  Call Extruder(271.09444)
  MoveL 11489 to (229.08, 163.95, 153.89) mm, rotated rx 180 ry 0 rz 180 deg; joints [-30.766, 12.961, 71.357, 80.556, 31.236, -78.992]
  MoveL 11490 to (229.08, 163.95, 153.89) mm, rotated rx 180 ry 0 rz 180 deg; joints [-30.766, 12.961, 71.357, 80.556, 31.236, -78.992]
  Call Extruder(271.20816)
  MoveL 11491 to (228.87, 164, 153.89) mm, rotated rx 180 ry 0 rz 180 deg; joints [-30.781, 12.934, 71.389, 80.571, 31.249, -79.007]
  MoveL 11492 to (228.87, 164, 153.89) mm, rotated rx 180 ry 0 rz 180 deg; joints [-30.781, 12.934, 71.389, 80.571, 31.249, -79.007]
  Call Extruder(271.33358)
  MoveL 11493 to (228.65, 164.04, 153.89) mm, rotated rx -180 ry 0 rz 180 deg; joints [-30.797, 12.904, 71.425, 80.587, 31.264, -79.024]
  MoveL 11494 to (228.65, 164.04, 153.89) mm, rotated rx -180 ry 0 rz 180 deg; joints [-30.797, 12.904, 71.425, 80.587, 31.264, -79.024]
  Call Extruder(271.47056)
  MoveL 11495 to (228.4, 164.09, 153.89) mm, rotated rx 180 ry 0 rz -180 deg; joints [-30.815, 12.872, 71.464, 80.604, 31.281, -79.042]
  MoveL 11496 to (228.4, 164.09, 153.89) mm, rotated rx 180 ry 0 rz -180 deg; joints [-30.815, 12.872, 71.464, 80.604, 31.281, -79.042]
  Call Extruder(271.60692)
  MoveL 11497 to (228.15, 164.14, 153.89) mm, rotated rx -180 ry 0 rz 180 deg; joints [-30.832, 12.839, 71.504, 80.622, 31.297, -79.06]
  MoveL 11498 to (228.15, 164.14, 153.89) mm, rotated rx -180 ry 0 rz 180 deg; joints [-30.832, 12.839, 71.504, 80.622, 31.297, -79.06]
  Call Extruder(271.74268)
  MoveL 11499 to (227.9, 164.19, 153.89) mm, rotated rx 180 ry 0 rz 180 deg; joints [-30.85, 12.806, 71.543, 80.639, 31.313, -79.079]
  MoveL 11500 to (227.9, 164.19, 153.89) mm, rotated rx 180 ry 0 rz 180 deg; joints [-30.85, 12.806, 71.543, 80.639, 31.313, -79.079]
  Call Extruder(271.87783)
  MoveL 11501 to (227.65, 164.24, 153.89) mm, rotated rx 180 ry 0 rz 180 deg; joints [-30.868, 12.773, 71.583, 80.656, 31.329, -79.097]
  MoveL 11502 to (227.65, 164.24, 153.89) mm, rotated rx 180 ry 0 rz 180 deg; joints [-30.868, 12.773, 71.583, 80.656, 31.329, -79.097]
  Call Extruder(272.01237)
  MoveL 11503 to (227.4, 164.29, 153.89) mm, rotated rx 180 ry 0 rz 180 deg; joints [-30.886, 12.74, 71.622, 80.674, 31.346, -79.115]
  MoveL 11504 to (227.4, 164.29, 153.89) mm, rotated rx 180 ry 0 rz 180 deg; joints [-30.886, 12.74, 71.622, 80.674, 31.346, -79.115]
  Call Extruder(272.14629)
  MoveL 11505 to (227.15, 164.34, 153.89) mm, rotated rx 180 ry 0 rz -180 deg; joints [-30.903, 12.708, 71.662, 80.691, 31.362, -79.133]
  MoveL 11506 to (227.15, 164.34, 153.89) mm, rotated rx 180 ry 0 rz -180 deg; joints [-30.903, 12.708, 71.662, 80.691, 31.362, -79.133]
  Call Extruder(272.29416)
  MoveL 11507 to (226.87, 164.39, 153.89) mm, rotated rx 180 ry 0 rz -180 deg; joints [-30.923, 12.671, 71.706, 80.71, 31.38, -79.154]
  MoveL 11508 to (226.87, 164.39, 153.89) mm, rotated rx 180 ry 0 rz -180 deg; joints [-30.923, 12.671, 71.706, 80.71, 31.38, -79.154]
  Call Extruder(272.45590)
  MoveL 11509 to (226.57, 164.44, 153.89) mm, rotated rx 180 ry 0 rz 180 deg; joints [-30.943, 12.63, 71.756, 80.731, 31.399, -79.176]
  MoveL 11510 to (226.57, 164.44, 153.89) mm, rotated rx 180 ry 0 rz 180 deg; joints [-30.943, 12.63, 71.756, 80.731, 31.399, -79.176]
  Call Extruder(272.61691)
  MoveL 11511 to (226.26, 164.49, 153.89) mm, rotated rx -180 ry 0 rz 180 deg; joints [-30.964, 12.588, 71.805, 80.752, 31.418, -79.198]
  MoveL 11512 to (226.26, 164.49, 153.89) mm, rotated rx -180 ry 0 rz 180 deg; joints [-30.964, 12.588, 71.805, 80.752, 31.418, -79.198]
  Call Extruder(272.77720)
  MoveL 11513 to (225.95, 164.54, 153.89) mm, rotated rx 180 ry 0 rz -180 deg; joints [-30.985, 12.547, 71.855, 80.773, 31.437, -79.22]
  MoveL 11514 to (225.95, 164.54, 153.89) mm, rotated rx 180 ry 0 rz -180 deg; joints [-30.985, 12.547, 71.855, 80.773, 31.437, -79.22]
  Call Extruder(272.93675)
  MoveL 11515 to (225.65, 164.58, 153.89) mm, rotated rx -180 ry 0 rz 180 deg; joints [-31.006, 12.506, 71.904, 80.794, 31.456, -79.242]
  MoveL 11516 to (225.65, 164.58, 153.89) mm, rotated rx -180 ry 0 rz 180 deg; joints [-31.006, 12.506, 71.904, 80.794, 31.456, -79.242]
  Call Extruder(273.09558)
  MoveL 11517 to (225.34, 164.63, 153.89) mm, rotated rx -180 ry 0 rz 180 deg; joints [-31.027, 12.465, 71.953, 80.814, 31.475, -79.264]
  MoveL 11518 to (225.34, 164.63, 153.89) mm, rotated rx -180 ry 0 rz 180 deg; joints [-31.027, 12.465, 71.953, 80.814, 31.475, -79.264]
  Call Extruder(273.27425)
  MoveL 11519 to (225, 164.68, 153.89) mm, rotated rx -180 ry 0 rz -180 deg; joints [-31.049, 12.418, 72.01, 80.838, 31.496, -79.289]
  MoveL 11520 to (225, 164.68, 153.89) mm, rotated rx -180 ry 0 rz -180 deg; joints [-31.049, 12.418, 72.01, 80.838, 31.496, -79.289]
  Call Extruder(273.47269)
  MoveL 11521 to (224.61, 164.73, 153.89) mm, rotated rx 180 ry 0 rz 180 deg; joints [-31.074, 12.364, 72.074, 80.864, 31.519, -79.316]
  MoveL 11522 to (224.61, 164.73, 153.89) mm, rotated rx 180 ry 0 rz 180 deg; joints [-31.074, 12.364, 72.074, 80.864, 31.519, -79.316]
  Call Extruder(273.67027)
  MoveL 11523 to (224.22, 164.77, 153.89) mm, rotated rx 180 ry 0 rz 180 deg; joints [-31.1, 12.311, 72.138, 80.89, 31.542, -79.344]
  MoveL 11524 to (224.22, 164.77, 153.89) mm, rotated rx 180 ry 0 rz 180 deg; joints [-31.1, 12.311, 72.138, 80.89, 31.542, -79.344]
  Call Extruder(273.86697)
  MoveL 11525 to (223.84, 164.82, 153.89) mm, rotated rx -180 ry 0 rz 180 deg; joints [-31.125, 12.258, 72.202, 80.915, 31.565, -79.371]
  MoveL 11526 to (223.84, 164.82, 153.89) mm, rotated rx -180 ry 0 rz 180 deg; joints [-31.125, 12.258, 72.202, 80.915, 31.565, -79.371]
  Call Extruder(274.06281)
  MoveL 11527 to (223.45, 164.86, 153.89) mm, rotated rx 180 ry 0 rz -180 deg; joints [-31.15, 12.204, 72.265, 80.941, 31.588, -79.398]
  MoveL 11528 to (223.45, 164.86, 153.89) mm, rotated rx 180 ry 0 rz -180 deg; joints [-31.15, 12.204, 72.265, 80.941, 31.588, -79.398]
  Call Extruder(274.35817)
  MoveL 11529 to (222.86, 164.91, 153.89) mm, rotated rx 180 ry 0 rz 180 deg; joints [-31.186, 12.122, 72.364, 80.979, 31.621, -79.44]
  MoveL 11530 to (222.86, 164.91, 153.89) mm, rotated rx 180 ry 0 rz 180 deg; joints [-31.186, 12.122, 72.364, 80.979, 31.621, -79.44]
  Call Extruder(274.65220)
  MoveL 11531 to (222.27, 164.95, 153.89) mm, rotated rx 180 ry 0 rz 180 deg; joints [-31.222, 12.039, 72.463, 81.018, 31.654, -79.48]
  MoveL 11532 to (222.27, 164.95, 153.89) mm, rotated rx 180 ry 0 rz 180 deg; joints [-31.222, 12.039, 72.463, 81.018, 31.654, -79.48]
  Call Extruder(274.94489)
  MoveL 11533 to (221.68, 165, 153.89) mm, rotated rx -180 ry 0 rz 180 deg; joints [-31.258, 11.956, 72.562, 81.056, 31.687, -79.521]
  MoveL 11534 to (221.68, 165, 153.89) mm, rotated rx -180 ry 0 rz 180 deg; joints [-31.258, 11.956, 72.562, 81.056, 31.687, -79.521]
  Call Extruder(275.51834)
  MoveL 11535 to (220.52, 165.05, 153.89) mm, rotated rx 180 ry 0 rz 180 deg; joints [-31.326, 11.789, 72.76, 81.13, 31.749, -79.601]
  MoveL 11536 to (220.52, 165.05, 153.89) mm, rotated rx 180 ry 0 rz 180 deg; joints [-31.326, 11.789, 72.76, 81.13, 31.749, -79.601]
  Call Extruder(276.23235)
  MoveL 11537 to (219.06, 165.09, 153.89) mm, rotated rx 180 ry 0 rz -180 deg; joints [-31.409, 11.579, 73.01, 81.221, 31.825, -79.699]
  Call Extruder(393.07903)
  MoveL 11538 to (-19.06, 165.09, 153.89) mm, rotated rx -180 ry 0 rz 180 deg; joints [-51.475, -16.768, 100.178, 84.78, 51.776, -81.601]
  Call Extruder(393.50763)
  MoveL 11539 to (-19.94, 165.07, 153.89) mm, rotated rx 180 ry 0 rz 180 deg; joints [-51.582, -16.85, 100.239, 84.782, 51.884, -81.585]
  MoveL 11540 to (-19.94, 165.07, 153.89) mm, rotated rx 180 ry 0 rz 180 deg; joints [-51.582, -16.85, 100.239, 84.782, 51.884, -81.585]
  Call Extruder(394.08108)
  MoveL 11541 to (-21.1, 165.03, 153.89) mm, rotated rx 180 ry 0 rz 180 deg; joints [-51.722, -16.963, 100.321, 84.785, 52.025, -81.562]
  MoveL 11542 to (-21.1, 165.03, 153.89) mm, rotated rx 180 ry 0 rz 180 deg; joints [-51.722, -16.963, 100.321, 84.785, 52.025, -81.562]
  Call Extruder(394.51538)
  MoveL 11543 to (-21.97, 164.98, 153.89) mm, rotated rx 180 ry 0 rz 180 deg; joints [-51.827, -17.048, 100.383, 84.786, 52.131, -81.545]
  MoveL 11544 to (-21.97, 164.98, 153.89) mm, rotated rx 180 ry 0 rz 180 deg; joints [-51.827, -17.048, 100.383, 84.786, 52.131, -81.545]
  Call Extruder(394.80941)
  MoveL 11545 to (-22.56, 164.93, 153.89) mm, rotated rx -180 ry 0 rz -180 deg; joints [-51.897, -17.108, 100.426, 84.786, 52.201, -81.532]
  MoveL 11546 to (-22.56, 164.93, 153.89) mm, rotated rx -180 ry 0 rz -180 deg; joints [-51.897, -17.108, 100.426, 84.786, 52.201, -81.532]
  Call Extruder(395.10477)
  MoveL 11547 to (-23.15, 164.89, 153.89) mm, rotated rx 180 ry 0 rz -180 deg; joints [-51.966, -17.167, 100.469, 84.787, 52.271, -81.52]
  MoveL 11548 to (-23.15, 164.89, 153.89) mm, rotated rx 180 ry 0 rz -180 deg; joints [-51.966, -17.167, 100.469, 84.787, 52.271, -81.52]
  Call Extruder(395.35098)
  MoveL 11549 to (-23.64, 164.84, 153.89) mm, rotated rx 180 ry 0 rz 180 deg; joints [-52.023, -17.217, 100.505, 84.787, 52.329, -81.509]
  MoveL 11550 to (-23.64, 164.84, 153.89) mm, rotated rx 180 ry 0 rz 180 deg; joints [-52.023, -17.217, 100.505, 84.787, 52.329, -81.509]
  Call Extruder(395.54769)
  MoveL 11551 to (-24.03, 164.79, 153.89) mm, rotated rx 180 ry 0 rz 180 deg; joints [-52.067, -17.258, 100.535, 84.787, 52.374, -81.5]
  MoveL 11552 to (-24.03, 164.79, 153.89) mm, rotated rx 180 ry 0 rz 180 deg; joints [-52.067, -17.258, 100.535, 84.787, 52.374, -81.5]
  Call Extruder(395.74526)
  MoveL 11553 to (-24.42, 164.75, 153.89) mm, rotated rx -180 ry 0 rz 180 deg; joints [-52.112, -17.299, 100.564, 84.786, 52.419, -81.491]
  MoveL 11554 to (-24.42, 164.75, 153.89) mm, rotated rx -180 ry 0 rz 180 deg; joints [-52.112, -17.299, 100.564, 84.786, 52.419, -81.491]
  Call Extruder(395.94370)
  MoveL 11555 to (-24.8, 164.7, 153.89) mm, rotated rx 180 ry 0 rz 180 deg; joints [-52.156, -17.339, 100.594, 84.786, 52.464, -81.481]
  MoveL 11556 to (-24.8, 164.7, 153.89) mm, rotated rx 180 ry 0 rz 180 deg; joints [-52.156, -17.339, 100.594, 84.786, 52.464, -81.481]
  Call Extruder(396.14301)
  MoveL 11557 to (-25.19, 164.66, 153.89) mm, rotated rx 180 ry 0 rz -180 deg; joints [-52.2, -17.38, 100.623, 84.785, 52.509, -81.472]
  MoveL 11558 to (-25.19, 164.66, 153.89) mm, rotated rx 180 ry 0 rz -180 deg; joints [-52.2, -17.38, 100.623, 84.785, 52.509, -81.472]
  Call Extruder(396.30184)
  MoveL 11559 to (-25.5, 164.61, 153.89) mm, rotated rx 180 ry 0 rz 180 deg; joints [-52.235, -17.413, 100.647, 84.785, 52.543, -81.465]
  MoveL 11560 to (-25.5, 164.61, 153.89) mm, rotated rx 180 ry 0 rz 180 deg; joints [-52.235, -17.413, 100.647, 84.785, 52.543, -81.465]
  Call Extruder(396.46140)
  MoveL 11561 to (-25.8, 164.56, 153.89) mm, rotated rx 180 ry 0 rz 180 deg; joints [-52.269, -17.447, 100.671, 84.784, 52.578, -81.457]
  MoveL 11562 to (-25.8, 164.56, 153.89) mm, rotated rx 180 ry 0 rz 180 deg; joints [-52.269, -17.447, 100.671, 84.784, 52.578, -81.457]
  Call Extruder(396.62169)
  MoveL 11563 to (-26.11, 164.51, 153.89) mm, rotated rx 180 ry 0 rz 180 deg; joints [-52.303, -17.48, 100.695, 84.783, 52.612, -81.449]
  MoveL 11564 to (-26.11, 164.51, 153.89) mm, rotated rx 180 ry 0 rz 180 deg; joints [-52.303, -17.48, 100.695, 84.783, 52.612, -81.449]
  Call Extruder(396.78271)
  MoveL 11565 to (-26.41, 164.46, 153.89) mm, rotated rx -180 ry 0 rz 180 deg; joints [-52.337, -17.514, 100.719, 84.782, 52.647, -81.441]
  MoveL 11566 to (-26.41, 164.46, 153.89) mm, rotated rx -180 ry 0 rz 180 deg; joints [-52.337, -17.514, 100.719, 84.782, 52.647, -81.441]
  Call Extruder(396.94445)
  MoveL 11567 to (-26.72, 164.41, 153.89) mm, rotated rx 180 ry 0 rz -180 deg; joints [-52.371, -17.547, 100.743, 84.782, 52.681, -81.433]
  MoveL 11568 to (-26.72, 164.41, 153.89) mm, rotated rx 180 ry 0 rz -180 deg; joints [-52.371, -17.547, 100.743, 84.782, 52.681, -81.433]
  Call Extruder(397.10692)
  MoveL 11569 to (-27.02, 164.37, 153.89) mm, rotated rx 180 ry 0 rz 180 deg; joints [-52.405, -17.58, 100.767, 84.781, 52.716, -81.425]
  MoveL 11570 to (-27.02, 164.37, 153.89) mm, rotated rx 180 ry 0 rz 180 deg; joints [-52.405, -17.58, 100.767, 84.781, 52.716, -81.425]
  Call Extruder(397.24085)
  MoveL 11571 to (-27.27, 164.32, 153.89) mm, rotated rx -180 ry 0 rz -180 deg; joints [-52.432, -17.609, 100.788, 84.78, 52.743, -81.418]
  MoveL 11572 to (-27.27, 164.32, 153.89) mm, rotated rx -180 ry 0 rz -180 deg; joints [-52.432, -17.609, 100.788, 84.78, 52.743, -81.418]
  Call Extruder(397.37538)
  MoveL 11573 to (-27.52, 164.27, 153.89) mm, rotated rx 180 ry 0 rz 180 deg; joints [-52.459, -17.637, 100.808, 84.779, 52.771, -81.411]
  MoveL 11574 to (-27.52, 164.27, 153.89) mm, rotated rx 180 ry 0 rz 180 deg; joints [-52.459, -17.637, 100.808, 84.779, 52.771, -81.411]
  Call Extruder(397.51053)
  MoveL 11575 to (-27.77, 164.22, 153.89) mm, rotated rx 180 ry 0 rz 180 deg; joints [-52.486, -17.665, 100.828, 84.778, 52.798, -81.404]
  MoveL 11576 to (-27.77, 164.22, 153.89) mm, rotated rx 180 ry 0 rz 180 deg; joints [-52.486, -17.665, 100.828, 84.778, 52.798, -81.404]
  Call Extruder(397.64629)
  MoveL 11577 to (-28.02, 164.17, 153.89) mm, rotated rx 180 ry 0 rz -180 deg; joints [-52.513, -17.693, 100.848, 84.777, 52.825, -81.397]
  MoveL 11578 to (-28.02, 164.17, 153.89) mm, rotated rx 180 ry 0 rz -180 deg; joints [-52.513, -17.693, 100.848, 84.777, 52.825, -81.397]
  Call Extruder(397.78265)
  MoveL 11579 to (-28.27, 164.12, 153.89) mm, rotated rx 180 ry 0 rz 180 deg; joints [-52.54, -17.722, 100.869, 84.776, 52.853, -81.391]
  MoveL 11580 to (-28.27, 164.12, 153.89) mm, rotated rx 180 ry 0 rz 180 deg; joints [-52.54, -17.722, 100.869, 84.776, 52.853, -81.391]
  Call Extruder(397.86751)
  MoveL 11581 to (-28.42, 164.09, 153.89) mm, rotated rx -180 ry 0 rz 180 deg; joints [-52.556, -17.739, 100.881, 84.775, 52.87, -81.386]
  Set speed (130.0 mm/s)
  MoveL 11582 to (-31.76, 163.31, 153.89) mm, rotated rx 180 ry 0 rz 180 deg; joints [-52.91, -18.13, 101.16, 84.758, 53.229, -81.286]
  Call Extruder(395.86751)
  Set speed (40.0 mm/s)
  MoveL 11583 to (-31.76, 163.31, 153.89) mm, rotated rx 180 ry 0 rz 180 deg; joints [-52.91, -18.13, 101.16, 84.758, 53.229, -81.286]
  Set speed (1000.0 mm/s)
  Call Extruder(-1)
  MoveL 11584 to (-31.76, 163.31, 153.89) mm, rotated rx 180 ry 0 rz 180 deg; joints [-52.91, -18.13, 101.16, 84.758, 53.229, -81.286]
  Call Extruder(0.00000)
  Call M_RunCode(107)
  Call M_RunCode(104)
  Call M_RunCode(84)
  Call M_RunCode(140)

--- program Print3D (robot Denso VS-6577G-B) ---
  Smooth(1)
  Call M_RunCode(107)
  Call M_RunCode(104)
  Set speed (83.3 mm/s)
  Set speed (1000.0 mm/s)
  Set Ref.: Ref002
  Set Tool: nozzle
  Show nozzle
  MoveJ 1 to (0, 34.91, 105) mm, rotated rx 180 ry 0 rz 180 deg; joints [-47.898, 28.981, 154.135, 132.06, 92.089, -2.313]
  MoveL 2 to (0, 34.91, 105) mm, rotated rx 180 ry 0 rz 180 deg; joints [-47.898, 28.981, 154.135, 132.06, 92.089, -2.313]
  MoveL 3 to (0, 34.91, 5) mm, rotated rx 180 ry 0 rz 180 deg; joints [-47.898, 52.446, 146.262, 130.56, 102.419, -14.104]
  MoveL 4 to (0, 34.91, 5) mm, rotated rx 180 ry 0 rz 180 deg; joints [-47.898, 52.446, 146.262, 130.56, 102.419, -14.104]
  Call M_RunCode(109)
  Call M_RunCode(82)
  Call Extruder(0.00000)
  Set speed (130.0 mm/s)
  MoveL 5 to (0, 34.91, 22.22) mm, rotated rx 180 ry 0 rz 180 deg; joints [-47.898, 48.666, 147.922, 130.893, 101.034, -12.462]
  Call Extruder(-2.00000)
  Set speed (40.0 mm/s)
  MoveL 6 to (0, 34.91, 22.22) mm, rotated rx 180 ry 0 rz 180 deg; joints [-47.898, 48.666, 147.922, 130.893, 101.034, -12.462]
  Call Extruder(0.00000)
  Set speed (130.0 mm/s)
  MoveL 7 to (0, 34.91, 22.22) mm, rotated rx 180 ry 0 rz 180 deg; joints [-47.898, 48.666, 147.922, 130.893, 101.034, -12.462]
  Call Extruder(2.00000)
  Set speed (40.0 mm/s)
  MoveL 8 to (0, 34.91, 22.22) mm, rotated rx 180 ry 0 rz 180 deg; joints [-47.898, 48.666, 147.922, 130.893, 101.034, -12.462]
  Set speed (30.0 mm/s)
  MoveL 9 to (0, 34.91, 22.22) mm, rotated rx 180 ry 0 rz 180 deg; joints [-47.898, 48.666, 147.922, 130.893, 101.034, -12.462]
  Call Extruder(209.10557)
  MoveL 10 to (207.51, 34.91, 22.22) mm, rotated rx 180 ry 0 rz 180 deg; joints [-29.348, 52.122, 123.468, 150.579, 86.157, 2.165]
  Call Extruder(210.41057)
  MoveL 11 to (208.82, 34.98, 22.22) mm, rotated rx 180 ry 0 rz -180 deg; joints [-29.266, 52.176, 123.285, 150.657, 86.041, 2.222]
  Call Extruder(213.89122)
  MoveL 12 to (212.3, 35.26, 22.22) mm, rotated rx 180 ry 0 rz 180 deg; joints [-29.038, 52.32, 122.803, 150.874, 85.737, 2.372]
  Call Extruder(214.76022)
  MoveL 13 to (213.16, 35.34, 22.23) mm, rotated rx 180 ry 0 rz 180 deg; joints [-28.98, 52.356, 122.683, 150.929, 85.662, 2.408]
  Call Extruder(215.62924)
  MoveL 14 to (214.01, 35.53, 22.23) mm, rotated rx -180 ry 0 rz -180 deg; joints [-28.913, 52.389, 122.574, 150.993, 85.592, 2.44]
  Call Extruder(219.10988)
  MoveL 15 to (217.4, 36.34, 22.22) mm, rotated rx 180 ry 0 rz 180 deg; joints [-28.639, 52.52, 122.143, 151.256, 85.317, 2.564]
  Call Extruder(219.97888)
  MoveL 16 to (218.25, 36.56, 22.23) mm, rotated rx 180 ry 0 rz -180 deg; joints [-28.569, 52.552, 122.036, 151.323, 85.249, 2.594]
  Call Extruder(220.84782)
  MoveL 17 to (219.06, 36.88, 22.23) mm, rotated rx 180 ry 0 rz 180 deg; joints [-28.492, 52.581, 121.942, 151.398, 85.189, 2.619]
  Call Extruder(224.32848)
  MoveL 18 to (222.28, 38.21, 22.23) mm, rotated rx -180 ry 0 rz -180 deg; joints [-28.179, 52.695, 121.572, 151.702, 84.949, 2.714]
  Call Extruder(225.19749)
  MoveL 19 to (223.08, 38.56, 22.23) mm, rotated rx 180 ry 0 rz 180 deg; joints [-28.099, 52.723, 121.482, 151.778, 84.89, 2.737]
  Call Extruder(226.06647)
  MoveL 20 to (223.83, 39, 22.22) mm, rotated rx 180 ry 0 rz -180 deg; joints [-28.014, 52.747, 121.405, 151.862, 84.839, 2.754]
  Call Extruder(229.54713)
  MoveL 21 to (226.8, 40.82, 22.22) mm, rotated rx 180 ry 0 rz 180 deg; joints [-27.668, 52.841, 121.105, 152.2, 84.64, 2.82]
  Call Extruder(230.41613)
  MoveL 22 to (227.53, 41.29, 22.22) mm, rotated rx 180 ry 0 rz -180 deg; joints [-27.581, 52.863, 121.032, 152.285, 84.591, 2.835]
  Call Extruder(231.28508)
  MoveL 23 to (228.21, 41.85, 22.22) mm, rotated rx 180 ry 0 rz 180 deg; joints [-27.489, 52.881, 120.974, 152.376, 84.552, 2.845]
  Call Extruder(234.76575)
  MoveL 24 to (230.86, 44.11, 22.22) mm, rotated rx -180 ry 0 rz 180 deg; joints [-27.119, 52.951, 120.751, 152.74, 84.397, 2.88]
  Call Extruder(235.63479)
  MoveL 25 to (231.51, 44.69, 22.22) mm, rotated rx 180 ry 0 rz -180 deg; joints [-27.026, 52.968, 120.698, 152.832, 84.36, 2.887]
  Call Extruder(236.50375)
  MoveL 26 to (232.09, 45.34, 22.23) mm, rotated rx 180 ry 0 rz -180 deg; joints [-26.929, 52.98, 120.66, 152.927, 84.333, 2.89]
  Call Extruder(239.98454)
  MoveL 27 to (234.35, 47.99, 22.22) mm, rotated rx 180 ry 0 rz 180 deg; joints [-26.542, 53.025, 120.52, 153.312, 84.227, 2.895]
  Call Extruder(240.85339)
  MoveL 28 to (234.91, 48.67, 22.22) mm, rotated rx -180 ry 0 rz -180 deg; joints [-26.445, 53.035, 120.487, 153.408, 84.202, 2.895]
  Call Extruder(241.72239)
  MoveL 29 to (235.38, 49.4, 22.22) mm, rotated rx -180 ry 0 rz 180 deg; joints [-26.346, 53.04, 120.471, 153.507, 84.187, 2.89]
  Call Extruder(245.20303)
  MoveL 30 to (237.2, 52.37, 22.22) mm, rotated rx 180 ry 0 rz -180 deg; joints [-25.95, 53.058, 120.416, 153.903, 84.134, 2.866]
  Call Extruder(246.07200)
  MoveL 31 to (237.64, 53.12, 22.22) mm, rotated rx -180 ry 0 rz -180 deg; joints [-25.851, 53.061, 120.404, 154.002, 84.121, 2.859]
  Call Extruder(246.94105)
  MoveL 32 to (237.99, 53.92, 22.22) mm, rotated rx 180 ry 0 rz 180 deg; joints [-25.752, 53.059, 120.409, 154.102, 84.12, 2.848]
  Call Extruder(250.42170)
  MoveL 33 to (239.32, 57.14, 22.22) mm, rotated rx -180 ry 0 rz 180 deg; joints [-25.354, 53.049, 120.441, 154.502, 84.12, 2.797]
  Call Extruder(251.29060)
  MoveL 34 to (239.64, 57.95, 22.22) mm, rotated rx 180 ry 0 rz 180 deg; joints [-25.255, 53.046, 120.451, 154.602, 84.121, 2.784]
  Call Extruder(252.15951)
  MoveL 35 to (239.86, 58.8, 22.22) mm, rotated rx 180 ry 0 rz -180 deg; joints [-25.158, 53.038, 120.478, 154.701, 84.133, 2.766]
  Call Extruder(255.64017)
  MoveL 36 to (240.67, 62.19, 22.22) mm, rotated rx 180 ry 0 rz -180 deg; joints [-24.767, 53, 120.596, 155.096, 84.188, 2.692]
  Call Extruder(256.50930)
  MoveL 37 to (240.86, 63.04, 22.22) mm, rotated rx -180 ry 0 rz 180 deg; joints [-24.67, 52.99, 120.628, 155.195, 84.203, 2.673]
  Call Extruder(257.37833)
  MoveL 38 to (240.94, 63.9, 22.22) mm, rotated rx 180 ry 0 rz -180 deg; joints [-24.576, 52.975, 120.676, 155.291, 84.228, 2.65]
  Call Extruder(260.85898)
  MoveL 39 to (241.22, 67.38, 22.22) mm, rotated rx 180 ry 0 rz 180 deg; joints [-24.2, 52.912, 120.876, 155.674, 84.336, 2.555]
  Call Extruder(262.16396)
  MoveL 40 to (241.29, 68.69, 22.22) mm, rotated rx -180 ry 0 rz 180 deg; joints [-24.06, 52.887, 120.956, 155.817, 84.38, 2.518]
  Call Extruder(324.66760)
  MoveL 41 to (241.29, 131.31, 22.22) mm, rotated rx 180 ry 0 rz 180 deg; joints [-17.173, 51.782, 124.636, 162.796, 86.578, 1.059]
  Call Extruder(325.97258)
  MoveL 42 to (241.22, 132.62, 22.23) mm, rotated rx -180 ry 0 rz -180 deg; joints [-17.025, 51.761, 124.71, 162.944, 86.625, 1.035]
  Call Extruder(329.45322)
  MoveL 43 to (240.94, 136.1, 22.23) mm, rotated rx 180 ry 0 rz 180 deg; joints [-16.634, 51.701, 124.918, 163.339, 86.761, 0.969]
  Call Extruder(330.32226)
  MoveL 44 to (240.86, 136.96, 22.22) mm, rotated rx -180 ry 0 rz -180 deg; joints [-16.537, 51.686, 124.972, 163.437, 86.796, 0.952]
  Call Extruder(331.19137)
  MoveL 45 to (240.67, 137.81, 22.22) mm, rotated rx 180 ry 0 rz -180 deg; joints [-16.445, 51.667, 125.041, 163.53, 86.842, 0.933]
  Call Extruder(334.67203)
  MoveL 46 to (239.86, 141.2, 22.23) mm, rotated rx -180 ry 0 rz -180 deg; joints [-16.078, 51.587, 125.323, 163.899, 87.031, 0.857]
  Call Extruder(335.54095)
  MoveL 47 to (239.64, 142.05, 22.22) mm, rotated rx 180 ry 0 rz -180 deg; joints [-15.988, 51.566, 125.396, 163.991, 87.08, 0.837]
  Call Extruder(336.40987)
  MoveL 48 to (239.32, 142.86, 22.22) mm, rotated rx 180 ry 0 rz 180 deg; joints [-15.904, 51.542, 125.482, 164.076, 87.138, 0.816]
  Call Extruder(339.89051)
  MoveL 49 to (237.99, 146.08, 22.23) mm, rotated rx 180 ry 0 rz -180 deg; joints [-15.57, 51.445, 125.833, 164.413, 87.378, 0.731]
  Call Extruder(340.75954)
  MoveL 50 to (237.64, 146.88, 22.22) mm, rotated rx 180 ry 0 rz 180 deg; joints [-15.488, 51.42, 125.922, 164.497, 87.439, 0.71]
  Call Extruder(341.62850)
  MoveL 51 to (237.2, 147.63, 22.22) mm, rotated rx -180 ry 0 rz 180 deg; joints [-15.413, 51.392, 126.024, 164.572, 87.509, 0.687]
  Call Extruder(345.10915)
  MoveL 52 to (235.38, 150.6, 22.22) mm, rotated rx 180 ry 0 rz 180 deg; joints [-15.12, 51.28, 126.436, 164.868, 87.794, 0.596]
  Call Extruder(345.97817)
  MoveL 53 to (234.91, 151.34, 22.22) mm, rotated rx 180 ry 0 rz 180 deg; joints [-15.048, 51.251, 126.54, 164.941, 87.867, 0.574]
  Call Extruder(346.84712)
  MoveL 54 to (234.35, 152.01, 22.22) mm, rotated rx -180 ry 0 rz 180 deg; joints [-14.986, 51.22, 126.654, 165.004, 87.947, 0.55]
  Call Extruder(350.32775)
  MoveL 55 to (232.09, 154.66, 22.23) mm, rotated rx 180 ry 0 rz 180 deg; joints [-14.741, 51.097, 127.117, 165.253, 88.272, 0.455]
  Call Extruder(351.19679)
  MoveL 56 to (231.51, 155.31, 22.23) mm, rotated rx 180 ry 0 rz 180 deg; joints [-14.681, 51.066, 127.233, 165.313, 88.355, 0.431]
  Call Extruder(352.06577)
  MoveL 57 to (230.86, 155.89, 22.22) mm, rotated rx -180 ry 0 rz 180 deg; joints [-14.632, 51.033, 127.358, 165.363, 88.443, 0.407]
  Call Extruder(355.54644)
  MoveL 58 to (228.21, 158.15, 22.22) mm, rotated rx 180 ry 0 rz -180 deg; joints [-14.441, 50.902, 127.86, 165.556, 88.801, 0.309]
  Call Extruder(356.41541)
  MoveL 59 to (227.53, 158.71, 22.22) mm, rotated rx 180 ry 0 rz 180 deg; joints [-14.395, 50.87, 127.986, 165.603, 88.892, 0.284]
  Call Extruder(357.28446)
  MoveL 60 to (226.8, 159.18, 22.23) mm, rotated rx 180 ry 0 rz -180 deg; joints [-14.36, 50.836, 128.118, 165.637, 88.987, 0.259]
  Call Extruder(360.76512)
  MoveL 61 to (223.83, 161, 22.22) mm, rotated rx 180 ry 0 rz 180 deg; joints [-14.23, 50.701, 128.649, 165.769, 89.37, 0.16]
  Call Extruder(361.63406)
  MoveL 62 to (223.08, 161.44, 22.23) mm, rotated rx -180 ry 0 rz -180 deg; joints [-14.199, 50.668, 128.782, 165.8, 89.467, 0.135]
  Call Extruder(362.50303)
  MoveL 63 to (222.28, 161.79, 22.23) mm, rotated rx -180 ry 0 rz -180 deg; joints [-14.181, 50.634, 128.918, 165.818, 89.566, 0.11]
  Call Extruder(365.98369)
  MoveL 64 to (219.06, 163.12, 22.23) mm, rotated rx -180 ry 0 rz -180 deg; joints [-14.116, 50.5, 129.464, 165.883, 89.965, 0.009]
  Call Extruder(366.85268)
  MoveL 65 to (218.25, 163.44, 22.22) mm, rotated rx 180 ry 0 rz 180 deg; joints [-14.102, 50.467, 129.6, 165.898, 90.065, -0.016]
  Call Extruder(367.72170)
  MoveL 66 to (217.4, 163.66, 22.22) mm, rotated rx 180 ry 0 rz 180 deg; joints [-14.101, 50.434, 129.737, 165.899, 90.166, -0.042]
  Call Extruder(371.20234)
  MoveL 67 to (214.01, 164.47, 22.23) mm, rotated rx 180 ry 0 rz 180 deg; joints [-14.106, 50.304, 130.285, 165.893, 90.572, -0.144]
  Call Extruder(372.07132)
  MoveL 68 to (213.16, 164.66, 22.22) mm, rotated rx 180 ry 0 rz 180 deg; joints [-14.11, 50.272, 130.422, 165.889, 90.673, -0.169]
  Call Extruder(372.94029)
  MoveL 69 to (212.3, 164.75, 22.22) mm, rotated rx 180 ry 0 rz 180 deg; joints [-14.126, 50.241, 130.556, 165.872, 90.773, -0.195]
  Call Extruder(376.42094)
  MoveL 70 to (208.82, 165.02, 22.22) mm, rotated rx -180 ry 0 rz -180 deg; joints [-14.203, 50.119, 131.093, 165.794, 91.175, -0.297]
  Call Extruder(377.28995)
  MoveL 71 to (207.95, 165.07, 22.22) mm, rotated rx 180 ry 0 rz 180 deg; joints [-14.224, 50.089, 131.226, 165.772, 91.275, -0.323]
  Call Extruder(377.72605)
  MoveL 72 to (207.51, 165.09, 22.22) mm, rotated rx 180 ry 0 rz -180 deg; joints [-14.236, 50.074, 131.293, 165.76, 91.325, -0.336]
  Call Extruder(592.33024)
  MoveL 73 to (-7.51, 165.09, 22.22) mm, rotated rx 180 ry 0 rz 180 deg; joints [-27.36, 52.911, 158.356, 148.809, 117.449, -15.593]
  Call Extruder(593.63529)
  MoveL 74 to (-8.82, 165.02, 22.22) mm, rotated rx 180 ry 0 rz 180 deg; joints [-27.524, 53.013, 158.475, 148.572, 117.594, -15.804]
  Call Extruder(597.11593)
  MoveL 75 to (-12.3, 164.74, 22.22) mm, rotated rx 180 ry 0 rz 180 deg; joints [-27.987, 53.287, 158.786, 147.907, 117.963, -16.387]
  Call Extruder(597.98490)
  MoveL 76 to (-13.16, 164.66, 22.22) mm, rotated rx -180 ry 0 rz 180 deg; joints [-28.108, 53.355, 158.862, 147.734, 118.051, -16.535]
  Call Extruder(598.85386)
  MoveL 77 to (-14.01, 164.47, 22.22) mm, rotated rx 180 ry 0 rz 180 deg; joints [-28.25, 53.419, 158.931, 147.542, 118.122, -16.689]
  Call Extruder(602.33452)
  MoveL 78 to (-17.4, 163.66, 22.22) mm, rotated rx 180 ry 0 rz 180 deg; joints [-28.842, 53.672, 159.199, 146.747, 118.387, -17.314]
  Call Extruder(603.20352)
  MoveL 79 to (-18.25, 163.44, 22.22) mm, rotated rx 180 ry 0 rz 180 deg; joints [-28.995, 53.735, 159.265, 146.543, 118.448, -17.473]
  Call Extruder(604.07254)
  MoveL 80 to (-19.06, 163.12, 22.22) mm, rotated rx 180 ry 0 rz 180 deg; joints [-29.167, 53.791, 159.321, 146.323, 118.49, -17.633]
  Call Extruder(607.55321)
  MoveL 81 to (-22.28, 161.79, 22.22) mm, rotated rx 180 ry 0 rz 180 deg; joints [-29.875, 54.01, 159.541, 145.423, 118.635, -18.279]
  Call Extruder(608.42217)
  MoveL 82 to (-23.08, 161.44, 22.22) mm, rotated rx -180 ry 0 rz 180 deg; joints [-30.056, 54.063, 159.594, 145.193, 118.665, -18.442]
  Call Extruder(609.29114)
  MoveL 83 to (-23.83, 161, 22.22) mm, rotated rx 180 ry 0 rz 180 deg; joints [-30.253, 54.108, 159.637, 144.953, 118.675, -18.602]
  Call Extruder(612.77178)
  MoveL 84 to (-26.8, 159.18, 22.23) mm, rotated rx -180 ry 0 rz 180 deg; joints [-31.057, 54.28, 159.802, 143.979, 118.689, -19.241]
  Call Extruder(613.64080)
  MoveL 85 to (-27.54, 158.71, 22.23) mm, rotated rx 180 ry 0 rz 180 deg; joints [-31.261, 54.321, 159.84, 143.733, 118.685, -19.401]
  Call Extruder(614.50982)
  MoveL 86 to (-28.21, 158.15, 22.22) mm, rotated rx -180 ry 0 rz 180 deg; joints [-31.477, 54.352, 159.869, 143.482, 118.661, -19.552]
  Call Extruder(617.99048)
  MoveL 87 to (-30.86, 155.89, 22.22) mm, rotated rx 180 ry 0 rz -180 deg; joints [-32.352, 54.466, 159.975, 142.473, 118.54, -20.151]
  Call Extruder(618.85941)
  MoveL 88 to (-31.51, 155.31, 22.23) mm, rotated rx 180 ry 0 rz 180 deg; joints [-32.573, 54.492, 159.999, 142.22, 118.503, -20.299]
  Call Extruder(619.72839)
  MoveL 89 to (-32.09, 154.66, 22.23) mm, rotated rx 180 ry 0 rz -180 deg; joints [-32.8, 54.507, 160.012, 141.968, 118.446, -20.434]
  Call Extruder(623.20904)
  MoveL 90 to (-34.35, 152.01, 22.23) mm, rotated rx 180 ry 0 rz -180 deg; joints [-33.715, 54.555, 160.056, 140.965, 118.194, -20.96]
  Call Extruder(624.07805)
  MoveL 91 to (-34.91, 151.34, 22.22) mm, rotated rx 180 ry 0 rz 180 deg; joints [-33.945, 54.564, 160.064, 140.716, 118.126, -21.088]
  Call Extruder(624.94703)
  MoveL 92 to (-35.38, 150.6, 22.23) mm, rotated rx 180 ry 0 rz -180 deg; joints [-34.175, 54.562, 160.062, 140.474, 118.039, -21.199]
  Call Extruder(628.42769)
  MoveL 93 to (-37.2, 147.63, 22.23) mm, rotated rx -180 ry 0 rz 180 deg; joints [-35.097, 54.541, 160.043, 139.517, 117.672, -21.624]
  Call Extruder(629.29668)
  MoveL 94 to (-37.64, 146.88, 22.23) mm, rotated rx 180 ry 0 rz 180 deg; joints [-35.327, 54.533, 160.036, 139.281, 117.576, -21.724]
  Call Extruder(630.16566)
  MoveL 95 to (-37.99, 146.08, 22.22) mm, rotated rx -180 ry 0 rz 180 deg; joints [-35.553, 54.513, 160.018, 139.058, 117.464, -21.806]
  Call Extruder(633.64631)
  MoveL 96 to (-39.32, 142.86, 22.23) mm, rotated rx -180 ry 0 rz -180 deg; joints [-36.447, 54.425, 159.937, 138.182, 117.002, -22.106]
  Call Extruder(634.51530)
  MoveL 97 to (-39.64, 142.05, 22.22) mm, rotated rx -180 ry 0 rz 180 deg; joints [-36.668, 54.4, 159.914, 137.969, 116.883, -22.175]
  Call Extruder(635.38427)
  MoveL 98 to (-39.86, 141.2, 22.23) mm, rotated rx 180 ry 0 rz -180 deg; joints [-36.88, 54.365, 159.881, 137.772, 116.752, -22.223]
  Call Extruder(638.86493)
  MoveL 99 to (-40.67, 137.81, 22.23) mm, rotated rx 180 ry 0 rz 180 deg; joints [-37.716, 54.214, 159.739, 137.007, 116.22, -22.387]
  Call Extruder(639.73393)
  MoveL 100 to (-40.86, 136.96, 22.23) mm, rotated rx 180 ry 0 rz 180 deg; joints [-37.921, 54.175, 159.701, 136.822, 116.085, -22.421]
  Call Extruder(640.60294)
  MoveL 101 to (-40.94, 136.1, 22.22) mm, rotated rx -180 ry 0 rz 180 deg; joints [-38.112, 54.126, 159.654, 136.657, 115.942, -22.434]
  Call Extruder(644.08358)
  MoveL 102 to (-41.22, 132.62, 22.22) mm, rotated rx 180 ry 0 rz 180 deg; joints [-38.861, 53.924, 159.456, 136.022, 115.367, -22.46]
  Call Extruder(645.38859)
  MoveL 103 to (-41.29, 131.31, 22.23) mm, rotated rx 180 ry 0 rz -180 deg; joints [-39.133, 53.845, 159.377, 135.796, 115.15, -22.458]
  Call Extruder(707.89230)
  MoveL 104 to (-41.29, 68.69, 22.23) mm, rotated rx 180 ry 0 rz -180 deg; joints [-49.612, 50.462, 154.512, 127.638, 105.877, -19.532]
  Call Extruder(709.19730)
  MoveL 105 to (-41.22, 67.38, 22.23) mm, rotated rx 180 ry 0 rz -180 deg; joints [-49.782, 50.405, 154.389, 127.512, 105.71, -19.429]
  Call Extruder(712.67795)
  MoveL 106 to (-40.94, 63.9, 22.23) mm, rotated rx -180 ry 0 rz -180 deg; joints [-50.212, 50.255, 154.052, 127.198, 105.273, -19.14]
  Call Extruder(713.54695)
  MoveL 107 to (-40.86, 63.04, 22.22) mm, rotated rx -180 ry 0 rz -180 deg; joints [-50.316, 50.218, 153.966, 127.123, 105.165, -19.065]
  Call Extruder(714.41596)
  MoveL 108 to (-40.67, 62.19, 22.23) mm, rotated rx -180 ry 0 rz 180 deg; joints [-50.4, 50.179, 153.873, 127.069, 105.058, -18.978]
  Call Extruder(717.89661)
  MoveL 109 to (-39.86, 58.8, 22.22) mm, rotated rx 180 ry 0 rz 180 deg; joints [-50.719, 50.026, 153.497, 126.869, 104.637, -18.62]
  Call Extruder(718.76559)
  MoveL 110 to (-39.64, 57.95, 22.22) mm, rotated rx 180 ry 0 rz -180 deg; joints [-50.794, 49.989, 153.401, 126.823, 104.533, -18.529]
  Call Extruder(719.63456)
  MoveL 111 to (-39.32, 57.14, 22.23) mm, rotated rx 180 ry 0 rz 180 deg; joints [-50.849, 49.95, 153.301, 126.798, 104.433, -18.428]
  Call Extruder(723.11522)
  MoveL 112 to (-37.99, 53.92, 22.23) mm, rotated rx 180 ry 0 rz 180 deg; joints [-51.053, 49.8, 152.895, 126.711, 104.036, -18.017]
  Call Extruder(723.98421)
  MoveL 113 to (-37.64, 53.12, 22.22) mm, rotated rx 180 ry 0 rz 180 deg; joints [-51.1, 49.764, 152.792, 126.692, 103.939, -17.914]
  Call Extruder(724.85321)
  MoveL 114 to (-37.2, 52.37, 22.22) mm, rotated rx -180 ry 0 rz 180 deg; joints [-51.126, 49.728, 152.687, 126.695, 103.846, -17.803]
  Call Extruder(728.33386)
  MoveL 115 to (-35.38, 49.4, 22.22) mm, rotated rx -180 ry 0 rz 180 deg; joints [-51.216, 49.587, 152.262, 126.717, 103.481, -17.357]
  Call Extruder(729.20284)
  MoveL 116 to (-34.91, 48.67, 22.23) mm, rotated rx -180 ry 0 rz 180 deg; joints [-51.235, 49.553, 152.155, 126.726, 103.391, -17.245]
  Call Extruder(730.07182)
  MoveL 117 to (-34.35, 47.99, 22.22) mm, rotated rx 180 ry 0 rz 180 deg; joints [-51.233, 49.52, 152.048, 126.754, 103.307, -17.129]
  Call Extruder(733.55248)
  MoveL 118 to (-32.09, 45.34, 22.23) mm, rotated rx 180 ry 0 rz 180 deg; joints [-51.212, 49.392, 151.614, 126.88, 102.977, -16.663]
  Call Extruder(734.42146)
  MoveL 119 to (-31.51, 44.69, 22.22) mm, rotated rx 180 ry 0 rz 180 deg; joints [-51.203, 49.361, 151.506, 126.914, 102.896, -16.547]
  Call Extruder(735.29045)
  MoveL 120 to (-30.86, 44.11, 22.22) mm, rotated rx 180 ry 0 rz -180 deg; joints [-51.175, 49.332, 151.398, 126.966, 102.822, -16.428]
  Call Extruder(738.77110)
  MoveL 121 to (-28.21, 41.85, 22.22) mm, rotated rx 180 ry 0 rz -180 deg; joints [-51.05, 49.22, 150.968, 127.187, 102.529, -15.957]
  Call Extruder(739.64010)
  MoveL 122 to (-27.54, 41.29, 22.23) mm, rotated rx 180 ry 0 rz 180 deg; joints [-51.016, 49.193, 150.86, 127.244, 102.457, -15.84]
  Call Extruder(740.50907)
  MoveL 123 to (-26.8, 40.82, 22.23) mm, rotated rx 180 ry 0 rz 180 deg; joints [-50.963, 49.168, 150.755, 127.319, 102.393, -15.724]
  Call Extruder(743.98973)
  MoveL 124 to (-23.83, 39, 22.22) mm, rotated rx 180 ry 0 rz 180 deg; joints [-50.742, 49.072, 150.338, 127.626, 102.14, -15.26]
  Call Extruder(744.85872)
  MoveL 125 to (-23.08, 38.56, 22.23) mm, rotated rx 180 ry 0 rz 180 deg; joints [-50.685, 49.049, 150.234, 127.704, 102.077, -15.146]
  Call Extruder(745.72772)
  MoveL 126 to (-22.28, 38.21, 22.22) mm, rotated rx 180 ry 0 rz 180 deg; joints [-50.61, 49.028, 150.135, 127.798, 102.023, -15.033]
  Call Extruder(749.20838)
  MoveL 127 to (-19.06, 36.88, 22.22) mm, rotated rx 180 ry 0 rz 180 deg; joints [-50.302, 48.948, 149.74, 128.181, 101.81, -14.588]
  Call Extruder(750.07736)
  MoveL 128 to (-18.25, 36.56, 22.23) mm, rotated rx 180 ry 0 rz 180 deg; joints [-50.223, 48.93, 149.642, 128.278, 101.757, -14.479]
  Call Extruder(750.94633)
  MoveL 129 to (-17.4, 36.34, 22.22) mm, rotated rx 180 ry 0 rz -180 deg; joints [-50.128, 48.913, 149.551, 128.39, 101.714, -14.373]
  Call Extruder(754.42699)
  MoveL 130 to (-14.01, 35.53, 22.23) mm, rotated rx 180 ry 0 rz 180 deg; joints [-49.744, 48.848, 149.188, 128.839, 101.542, -13.956]
  Call Extruder(755.29600)
  MoveL 131 to (-13.16, 35.34, 22.22) mm, rotated rx 180 ry 0 rz 180 deg; joints [-49.646, 48.833, 149.098, 128.952, 101.499, -13.853]
  Call Extruder(756.16500)
  MoveL 132 to (-12.3, 35.25, 22.22) mm, rotated rx -180 ry 0 rz 180 deg; joints [-49.535, 48.82, 149.017, 129.077, 101.466, -13.756]
  Call Extruder(759.64564)
  MoveL 133 to (-8.82, 34.98, 22.23) mm, rotated rx 180 ry 0 rz 180 deg; joints [-49.084, 48.77, 148.695, 129.582, 101.336, -13.374]
  Call Extruder(760.51461)
  MoveL 134 to (-7.95, 34.93, 22.23) mm, rotated rx 180 ry 0 rz 180 deg; joints [-48.971, 48.758, 148.615, 129.709, 101.304, -13.28]
  Call Extruder(760.95070)
  MoveL 135 to (-7.51, 34.91, 22.22) mm, rotated rx 180 ry 0 rz -180 deg; joints [-48.913, 48.752, 148.576, 129.773, 101.289, -13.234]
  Call Extruder(765.12213)
  MoveL 136 to (-3.33, 34.91, 22.22) mm, rotated rx 180 ry 0 rz 180 deg; joints [-48.345, 48.703, 148.214, 130.4, 101.151, -12.803]
  Call Extruder(763.12213)
  Set speed (40.0 mm/s)
  MoveL 137 to (-3.33, 34.91, 22.22) mm, rotated rx 180 ry 0 rz 180 deg; joints [-48.345, 48.703, 148.214, 130.4, 101.151, -12.803]
  Set speed (1000.0 mm/s)
  MoveL 138 to (-3.33, 34.91, 22.22) mm, rotated rx 180 ry 0 rz 180 deg; joints [-48.345, 48.703, 148.214, 130.4, 101.151, -12.803]
  MoveL 139 to (-3.33, 34.91, 122.23) mm, rotated rx 180 ry 0 rz 180 deg; joints [-48.345, 24.541, 155.335, 131.655, 89.917, 0.093]
  Call Extruder(0.00000)
  Call M_RunCode(104)
  Call M_RunCode(84)
  Call M_RunCode(140)

--- Python program Extruder ---
# This macro allows simulating a 3D printing extruder
# The macro will output spray gun statistics
#
# More information about the RoboDK API here:
# https://robodk.com/doc/en/RoboDK-API.html
# For more information visit:
# http://www.robodk.com/doc/en/PythonAPI/robolink.html
#
# Define the default action (0 to deactivate, +1 to activate, -1 to clear any spray gun simulation)
# Setting it to None will display a message
ACTION = None
# Check if we are running this program inside another program and passing arguments
import sys
if len(sys.argv) > 1:
    ACTION = float(sys.argv[1])
    # For faster speed: igone values greater than 0
    if ACTION > 0:
        quit()

from robolink import *    # API to communicate with RoboDK
from robodk import *      # basic matrix operations
RDK = Robolink()

# quit if we are not in simulation mode
if RDK.RunMode() != RUNMODE_SIMULATE:
    quit()

# Get any previously added spray gun simulations and display statistics (spray on the part vs spray falling out of the part)
existing_material_simulation = False
info, stats_data = RDK.Spray_GetStats()
if stats_data.size(1) > 0:
    print("Spray gun statistics:")
    print(info)
    print(stats_data.tr())
    existing_material_simulation = True
    # # Diplay statistics
    # RDK.ShowMessage("Material used: %.1f%%<br>Material waisted: %.1f%%<br>Total particles: %.1f" % (data[1,0],data[2,0],data[3,0]), True)
    # # Clear previous spray
    # RDK.Spray_Clear()

# If the default ACTION is None, display a message to activate/deactivate the spray gun
if ACTION is None:
    print('Note: This macro can be called as Extruder(0) to turn it ON or Extruder(-1) to turn it OFF')
    entry = mbox('Turn Extruder ON or OFF', ('On', '0'), ('Off', '-1'))
    if not entry:
        quit()
    ACTION = int(entry)

if ACTION < 0:
    # Turn material deposition off
    # Select Escape to delete existing material simulations
    #RDK.Spray_Clear()
    RDK.Spray_SetState(SPRAY_OFF)

elif ACTION >= 0:

    if existing_material_simulation:
        # Select Esc key to delete existing material simulations and force a new type of spray gun simulation
        RDK.Spray_SetState(SPRAY_ON)
        exit()


    # Create a new spray gun object in RoboDK for material deposition (3D printing simulation)
    # by using RDK.Spray_Add(tool, object, options_command, volume, geometry)
    # tool: tool item (TCP) to use
    # object: object to project the particles
    # options_command (optional): string to specify options. Example:
    #     STEP=AxB: Defines the grid to be projected 1x1 means only one line of particle projection (for example, for welding)
    #     PARTICLE: Defines the shape and size of particle (sphere or particle), unless a specific geometry is provided:
    #       a- SPHERE(radius, facets)
    #       b- SPHERE(radius, facets, scalex, scaley, scalez)
    #       b- CUBE(sizex, sizey, sizez)
    #     RAND=factor: Defines a random factor factor 0 means that the particles are not deposited randomly
    #     ELLYPSE: defines the volume as an ellypse (default)
    #     RECTANGLE: defines the volume as a rectangle
    #     PROJECT: project the particles to the surface (default) (for welding, painting or scanning)
    #     NO_PROJECT: does not project the particles to the surface (for example, for 3D printing)
    #
    # volume (optional): Matrix of parameters defining the volume of the spray gun
    # geometry (optional): Matrix of vertices defining the triangles.


    diameter = 22.225 # in mm
    detail = 8 # number of rings of detail to display the sphere
    scale = '1,1,0.5' # scale the particle in 0.5 along the tool Z axis (simulating gravity effect)
    options_command = "ELLYPSE NO_PROJECT PARTICLE=SPHERE(%.3f,%.0f,%s)" % (diameter, detail, scale) # simulate
    #options_command = "PARTICLE=CUBE(10,10,2) STEP=8x8"
    #options_command = "PARTICLE=SPHERE(4,8) STEP=8x8"
    #options_command = "PARTICLE=SPHERE(4,8,1,1,0.1) STEP=8x8 RAND=3"

    # Example commands for welding:
    # options_command = "PROJECT PARTICLE=SPHERE(4,8)"
    # options_command = PARTICLE=SPHERE(4,8) STEP=1x0

    tool = 0    # auto detect active tool
    obj = 0     # auto detect object in active reference frame

    # Material is deposited at 0,0,0 with respect to the TCP coordinates
    close_param = [0,0,0,  0,0,0,  0,0,0,     0.7,0.5,0.8,1] # color as RGBA
    far_param   = [0,0,0,  0,0,0,  0,0,0,     0.7,0.5,0.8,1] # color as RGBA
    volume = Mat([close_param, far_param])
    RDK.Spray_Add(tool, obj, options_command, volume.tr())
    RDK.Spray_SetState(SPRAY_ON)

--- Python program SimulateFinalResult ---
# This script will simulate the final result of the 3D printed part using the Spray function

# Or visit: http://www.robodk.com/doc/PythonAPI/
# Note: you do not need to keep a copy of this file, your python script is saved with the station
from robolink import *    # API to communicate with RoboDK
from robodk import *      # basic matrix operations


RENDER = True      # Set to False
STEP_MM = 2         # Detail step in MM for linear moves
STEP_DEG = 2        # Detail step in DEG for joint moves

# Start a connection with the RoboDK API
RDK = Robolink()

# Select the first/only robot in the cell:
program = RDK.ItemUserPick('Select a program to simulate', ITEM_TYPE_PROGRAM)
if not program.Valid():
    raise Exception("No program available")

# Get the robot
robot = RDK.Item('', ITEM_TYPE_ROBOT)
#robot = program.getLink(ITEM_TYPE_ROBOT) # available in newer versions
if not robot.Valid():
    raise Exception("No robot available")

progname = program.Name()
print("Using program %s" % progname)


# Get the program as a list of joint values
tool = robot.getLink(ITEM_TYPE_TOOL)
progok_jlist = program.InstructionListJoints(STEP_MM, STEP_DEG)
progok = progok_jlist[0] # progok: String that indicates if there are any issues with the program
jlist = progok_jlist[1]  # jlist: list of joints

# Check that the program is correct and has at least a movement
njoints = jlist.size(1)
if njoints < 1:
    raise Exception("Program %s has no movements" % name)

# Check if there are any issues with the program:
if progok != "Success":
    raise Exception("Problems with program %s: %s." %(name, progok))

# Reset any material deposition simulation
RDK.Spray_Clear()

robot.setPoseTool(tool)

# Start material deposition simulation according to the Extruder script
RDK.RunProgram('Extruder(0)')
# Alternatively:
#RDK.Item('Extruder', ITEM_TYPE_PYTHON).RunProgram([1])

if not RENDER:
    RDK.Render(False)

# Iterate through all joints in the matrix and check for collisions
njoints_all = jlist.size(1)
for i in range(njoints_all):
    ji = jlist[:,i].tolist()

    # Update the robot to a new position (it will create a new particle)
    robot.setJoints(ji)
    if not RENDER:
        # If Render is turned off (faster) update the position to draw a new particle
        RDK.Update()

    # Show a message in the RoboDK status bar from time to time
    if i % 10 == 0:
        msg = "Quick material deposition simulation for %s (%.1f %%)" % (progname, 100.0*(i/njoints_all))
        print(msg)
        RDK.ShowMessage(msg, False)

    # Render from time to time even if we have render deactivated
    if not RENDER and i % 500 == 0:
        RDK.Render()

RDK.Render(True)
msg = "Done"
print("Done")
RDK.ShowMessage(msg, False)
